FUNCTION_BLOCK FB_Axis_BaseUnit EXTENDS FB_BaseUnit IMPLEMENTS I_Axis_BaseUnit
VAR_INPUT
END_VAR
VAR_OUTPUT
END_VAR

VAR
	_Axis		: AXIS_REF;
	_MCMoveAbs	: MC_MoveAbsolute;
	_MCReset	: MC_Reset;
	_MCStop		: MC_Stop;
	_MCMoveVel	: MC_MoveVelocity;
	_MCMoveVel_2 : MC_MoveVelocity;
	_VelSwitchTrig : F_TRIG;
	_bVelSwitch : BOOL;
	_MCPower	: MC_Power;
	_MCJog		: MC_Jog;
	_MCHalt		: MC_Halt;
END_VAR

M_CyclicUpdate();

PROPERTY PUBLIC AxisActualVelocity : LREAL
GET
// Expose motion feedback without exposing AXIS_REF to Services.
AxisActualVelocity := _Axis.NcToPlc.ActVelo;
END_GET
END_PROPERTY

PROPERTY PUBLIC AxisHasJob : BOOL
GET
// Expose motion feedback without exposing AXIS_REF to Services.
AxisHasJob := _Axis.Status.HasJob;
END_GET
END_PROPERTY

PROPERTY PUBLIC AxisIsDisabled : BOOL
GET
// Treat an invalid Axis reference as unavailable to callers.
AxisIsDisabled := _Axis.Status.Disabled;
END_GET
END_PROPERTY

METHOD M_CyclicUpdate
VAR_INPUT
END_VAR
_MCPower(Axis:= _Axis,
			Enable:= TRUE,
			Enable_Positive:= TRUE,
			Enable_Negative:= TRUE,
			Override:= 100);
			
_MCReset(Axis:= _Axis);
_MCStop(Axis:= _Axis);
_MCMoveAbs(Axis:= _Axis);
_MCMoveVel(Axis:= _Axis);
_MCMoveVel_2(Axis:= _Axis);
_MCJog(Axis:= _Axis);
_MCHalt(Axis:= _Axis);

_Axis.ReadStatus();
END_METHOD

METHOD M_Halt : BOOL
VAR_INPUT
	OwnerId : T_ResourceOwnerId;
	Execute : BOOL;
	Deceleration : LREAL;
END_VAR
VAR_OUTPUT
	Done : BOOL;
	Error : BOOL;
END_VAR
M_Halt := FALSE;
Done := FALSE;
Error := FALSE;
IF NOT M_IsResourceOwner(OwnerId := OwnerId) THEN
	RETURN;
END_IF

_MCHalt.Execute := Execute;
_MCHalt.Deceleration := Deceleration;

Done := _MCHalt.Done;
Error := _MCHalt.Error;
M_Halt := TRUE;
END_METHOD

METHOD M_Jog : BOOL
VAR_INPUT
	OwnerId : T_ResourceOwnerId;
	JogForward : BOOL;
	JogBackwards : BOOL;
	Mode : E_JogMode;
	Position : LREAL;
	Velocity : LREAL;
	Acceleration : LREAL;
	Deceleration : LREAL;
END_VAR

VAR_OUTPUT
	Done : BOOL;
	Error : BOOL;
	ErrorId : UDINT;
END_VAR
// Ignore commands from Services that do not own this BaseUnit.
M_Jog := FALSE;
Done := FALSE;
Error := FALSE;
ErrorId := 0;
IF NOT M_IsResourceOwner(OwnerId := OwnerId) THEN
	RETURN;
END_IF

_MCJog.JogForward := JogForward;
_MCJog.JogBackwards := JogBackwards;
_MCJog.Mode := Mode;
_MCJog.Position := Position;
_MCJog.Velocity := Velocity;
_MCJog.Acceleration := Acceleration;
_MCJog.Deceleration := Deceleration;

Done := _MCJog.Done;
Error := _MCJog.Error;
ErrorId := _MCJog.ErrorId;
M_Jog := TRUE;
END_METHOD

METHOD M_MoveAbs : BOOL
VAR_INPUT
	OwnerId : T_ResourceOwnerId;
	Execute : BOOL;
	Position : LREAL;
	Velocity : LREAL;
	Acceleration : LREAL;
	Deceleration : LREAL;
END_VAR

VAR_OUTPUT
	Done : BOOL;
	Error : BOOL;
	ErrorId : UDINT;
END_VAR
// Ignore commands from Services that do not own this BaseUnit.
M_MoveAbs := FALSE;
Done := FALSE;
Error := FALSE;
ErrorId := 0;
IF NOT M_IsResourceOwner(OwnerId := OwnerId) THEN
	RETURN;
END_IF

_MCMoveAbs.Execute := Execute;
_MCMoveAbs.Position := Position;
_MCMoveAbs.Velocity := Velocity;
_MCMoveAbs.Acceleration := Acceleration;
_MCMoveAbs.Deceleration := Deceleration;

Done := _MCMoveAbs.Done;
Error := _MCMoveAbs.Error;
ErrorId := _MCMoveAbs.ErrorId;
M_MoveAbs := TRUE;
END_METHOD

METHOD M_MoveVel : BOOL
VAR_INPUT
	OwnerId : T_ResourceOwnerId;
	Execute : BOOL;
	Direction : MC_Direction;
	Velocity : LREAL;
	Acceleration : LREAL;
	Deceleration : LREAL;
END_VAR

VAR_OUTPUT
	InVelocity : BOOL;
	Error : BOOL;
END_VAR
// Ignore commands from Services that do not own this BaseUnit.
M_MoveVel := FALSE;
InVelocity := FALSE;
Error := FALSE;
IF NOT M_IsResourceOwner(OwnerId := OwnerId) THEN
	RETURN;
END_IF

// Clear input
IF Execute = FALSE THEN
	_MCMoveVel.Execute := FALSE;
	_MCMoveVel_2.Execute := FALSE;
END_IF

// Switch MoveVelocity when falling trig
_VelSwitchTrig(CLK:= Execute, Q=> );
IF _VelSwitchTrig.Q THEN
	_bVelSwitch := NOT _bVelSwitch;
END_IF

IF _bVelSwitch THEN
	_MCMoveVel.Execute := Execute;
	_MCMoveVel.Direction := Direction;
	_MCMoveVel.Velocity := Velocity;
	_MCMoveVel.Acceleration := Acceleration;
	_MCMoveVel.Deceleration := Deceleration;
	InVelocity := _MCMoveVel.InVelocity;
	Error := _MCMoveVel.Error;
ELSE
	_MCMoveVel_2.Execute := Execute;
	_MCMoveVel_2.Direction := Direction;
	_MCMoveVel_2.Velocity := Velocity;
	_MCMoveVel_2.Acceleration := Acceleration;
	_MCMoveVel_2.Deceleration := Deceleration;
	InVelocity := _MCMoveVel_2.InVelocity;
	Error := _MCMoveVel_2.Error;
	
END_IF

M_MoveVel := TRUE;
END_METHOD

METHOD M_Reset : BOOL
VAR_INPUT
	OwnerId : T_ResourceOwnerId;
	Execute : BOOL;
END_VAR

VAR_OUTPUT
	Done : BOOL;
	Error : BOOL;
	ErrorId : UDINT;
END_VAR
// Ignore commands from Services that do not own this BaseUnit.
M_Reset := FALSE;
Done := FALSE;
Error := FALSE;
ErrorId := 0;
IF NOT M_IsResourceOwner(OwnerId := OwnerId) THEN
	RETURN;
END_IF

_MCReset.Execute := Execute;

Done := _MCReset.Done;
Error := _MCReset.Error;
ErrorId := _MCReset.ErrorId;
M_Reset := TRUE;
END_METHOD

METHOD M_Stop : BOOL
VAR_INPUT
	OwnerId : T_ResourceOwnerId;
	Execute : BOOL;
	Deceleration : LREAL;
END_VAR

VAR_OUTPUT
	Done : BOOL;
	Error : BOOL;
	ErrorId : UDINT;
END_VAR
M_Stop := FALSE;
Done := FALSE;
Error := FALSE;
ErrorId := 0;
IF NOT M_IsResourceOwner(OwnerId := OwnerId) THEN
	RETURN;
END_IF

_MCStop.Execute := Execute;
_MCStop.Deceleration := Deceleration;

Done := _MCStop.Done;
Error := _MCStop.Error;
ErrorId := _MCStop.ErrorId;
M_Stop := TRUE;
END_METHOD

END_FUNCTION_BLOCK

(* stored: Version 1.1.0.1, ProductVersion 3.1.4026.18
   POU FB_Axis_BaseUnit: Id {28a42f80-195a-4223-a1bf-e623b7d6079c}, SpecialFunc None
   Property AxisActualVelocity: Id {777cc680-8953-4809-acb4-3307920aad6a}
   Get Get: Id {6b9ebc4e-1a8b-44c2-b05b-897b536b184f}
   Property AxisHasJob: Id {309289ed-139a-40cf-bb0b-b305e6a96468}
   Get Get: Id {6e6f9de3-535f-4e83-8a40-0db1c9ce0dbc}
   Property AxisIsDisabled: Id {24be025b-4296-4b69-8f78-3579130a7e1b}
   Get Get: Id {108a228b-e076-4883-9069-662ffabb72c6}
   Method M_CyclicUpdate: Id {40d31be8-e262-49a2-98a0-53468206e8c7}
   Method M_Halt: Id {99020f71-ff22-43ce-a9cc-2f51d191b702}
   Method M_Jog: Id {dc88b92a-725e-4df4-aa19-7fa274329a3a}
   Method M_MoveAbs: Id {12c6fae0-35a4-42f7-a077-cdf0cbcaba8d}
   Method M_MoveVel: Id {2b358657-cee5-4620-ae42-419450a93b24}
   Method M_Reset: Id {73fb1eb2-f7fa-423b-ae99-c942ced73b28}
   Method M_Stop: Id {2df51e0d-c316-436a-9fe7-294a4bc52bdf} *)
